// Mitsubishi GX Works2 project: Group12_PLC s (3)   PLC: FX3G

// global labels: Global1
VAR_GLOBAL
  startSwitch AT X007 : BOOL;
  initBisuit AT D1100 : REAL;
END_VAR
VAR_GLOBAL CONSTANT
  sixBis : REAL := 6.0;
END_VAR
VAR_GLOBAL
  enoughBuscuits AT M0 : BOOL;
  initCream AT D1102 : REAL;
END_VAR
VAR_GLOBAL CONSTANT
  threeHunCream : REAL := 300.0;
END_VAR
VAR_GLOBAL
  enoughCream AT M1 : BOOL;
  initChoclate AT D1104 : REAL;
END_VAR
VAR_GLOBAL CONSTANT
  twofourtyCho : REAL := 240.0;
END_VAR
VAR_GLOBAL
  enoughCoclate AT M2 : BOOL;
  startWday AT Y007 : BOOL;
  storeBuscuit AT D1106 : REAL;
  storeCream AT D1108 : REAL;
  storeChoclate AT D1110 : REAL;
  WD_started AT M40 : BOOL;
  FP_QA AT Y003 : BOOL;
  closeDay_HL AT M3 : BOOL;
  check AT M4 : BOOL;
  blink AT M4 : BOOL;
  activeDay AT Y007 : BOOL;
  stop3sec AT M5 : BOOL;
  activeDay_LI AT Y007 : BOOL;
  endBlink AT M6 : BOOL;
  finishing AT M60 : BOOL;
END_VAR
VAR_GLOBAL CONSTANT
  zeroCon : REAL;
END_VAR
VAR_GLOBAL
  stCounter AT CC1 : BOOL;
  scndCounter AT CC2 : BOOL;
  perfusion AT D1111 : REAL;
  Cream_perfusion AT D1112 : REAL;
  surfaceA AT D1114 : REAL;
  surfaceb AT D1116 : REAL;
  readyKrimbo AT D1118 : REAL;
  enoughBuscuitsTo_GoOn AT M10 : BOOL;
  enoughCreamTo_GoOn AT M11 : BOOL;
  enoughCoclateTo_GoOn AT M12 : BOOL;
  enoughStore AT M80 : BOOL;
  Ziluf_switch AT X011 : BOOL;
  ZilufContiner AT D1112 : REAL;
  moveToZiluf AT M90 : BOOL;
  moveTo_Ziluf AT M90 : BOOL;
  Machinestart_switchA AT X010 : BOOL;
  Carambosurface AT X001 : BOOL;
  Sprinkling_performed AT X003 : BOOL;
  TempAbove30 AT X030 : BOOL;
  TempLower15 AT X015 : BOOL;
  Sprinkling_isOn AT Y010 : BOOL;
  Machine_lampA AT Y004 : BOOL;
  faultIs_detected AT X002 : BOOL;
  stopMachine AT X005 : BOOL;
  ziluf_isOn AT Y010 : BOOL;
  krimboSurface AT X001 : BOOL;
END_VAR
VAR_GLOBAL CONSTANT
  subCream300 : REAL := 300.0;
  subBisctuit : REAL := 6.0;
END_VAR
VAR_GLOBAL
  Machine_lampAOn AT Y004 : BOOL;
  perfusion_performed AT X003 : BOOL;
  MachineA AT Y004 : BOOL;
  MachineA_off AT Y004 : BOOL;
  Machine_lampAoff AT X005 : BOOL;
  imageProcessing AT X003 : BOOL;
  perfusion_lampA AT Y004 : BOOL;
  perfusion_lampAOn AT Y004 : BOOL;
  perfusion_lampAoff AT X005 : BOOL;
  perfusion_switchA AT X010 : BOOL;
  Transportation AT M13 : BOOL;
  Timer4 AT TC4 : BOOL;
END_VAR
VAR_GLOBAL CONSTANT
  four_seconds : INT := 40;
END_VAR
VAR_GLOBAL
  output_Timer4 AT TS4 : BOOL;
  output_Timer3 AT TS4 : BOOL;
  output_Timer1 AT TS1 : BOOL;
  blinking_Input AT M14 : BOOL;
END_VAR
VAR_GLOBAL CONSTANT
  half_Second : INT := 5;
END_VAR
VAR_GLOBAL
  Timer2 AT TC0 : BOOL;
  Timer0 AT TC0 : BOOL;
  output_Timer0 AT TS0 : BOOL;
  Trans_Lamp0 AT Y000 : BOOL;
  Timer1 AT TC1 : BOOL;
  Trans_Lamp1 AT Y001 : BOOL;
  end_Tranportation AT M15 : BOOL;
  endTranportation AT M15 : BOOL;
  startFroasting AT X006 : BOOL;
  start_Froasting AT X006 : BOOL;
  AnalogInput1 AT D8280 : INT;
  save_Analog_Value AT D1114 : INT;
END_VAR
VAR_GLOBAL CONSTANT
  realUnit : INT := 400;
  ConstFive : INT := 5;
END_VAR
VAR_GLOBAL
  normalFroasting AT M16 : BOOL;
END_VAR
VAR_GLOBAL CONSTANT
  ConstTen : INT := 10;
END_VAR
VAR_GLOBAL
  less_thanTen : BOOL;
END_VAR
VAR_GLOBAL CONSTANT
  ConstSex : INT := 6;
  ConstSix : INT := 6;
END_VAR
VAR_GLOBAL
  doubleFroasting AT M17 : BOOL;
END_VAR
VAR_GLOBAL CONSTANT
  Chocolate_normalAmount : REAL := 120.0;
  Chocolate_normalAmount120 : REAL := 120.0;
END_VAR
VAR_GLOBAL
  Chocolate_in_process AT D1116 : REAL;
END_VAR
VAR_GLOBAL CONSTANT
  Chocolate_normalAmount240 : REAL := 240.0;
  Chocolate_doubleAmount240 : REAL := 240.0;
END_VAR
VAR_GLOBAL
  Finished_normalChocolateProcess AT M18 : BOOL;
  Finished_doubleChocolateProcess AT M19 : BOOL;
  Timer5 AT TC5 : BOOL;
END_VAR
VAR_GLOBAL CONSTANT
  five_seconds : INT := 50;
END_VAR
VAR_GLOBAL
  Froasting_Timer AT TS5 : BOOL;
  Froasting_Lamp AT Y003 : BOOL;
  startPackaging_krimbo AT X000 : BOOL;
  startCounter5_krimpo AT CC5 : BOOL;
END_VAR
VAR_GLOBAL CONSTANT
  Five_units : INT := 5;
END_VAR
VAR_GLOBAL
  finish_counter AT CS1 : BOOL;
END_VAR
VAR_GLOBAL CONSTANT
  six_units : INT := 6;
END_VAR
VAR_GLOBAL
  end_counting AT CC22 : BOOL;
  finish_packaging AT M20 : BOOL;
  end_countingPackaged AT CC6 : BOOL;
  end_packaging AT CS2 : BOOL;
  packagingLamp AT Y002 : BOOL;
  Add_6Krimbo AT D8280 : INT;
  krimbos_quantity AT D1118 : INT;
  start_WorkDay AT X007 : BOOL;
  end_DayBlink AT M66 : BOOL;
  blink_Seconds AT TC3 : BOOL;
END_VAR
VAR_GLOBAL CONSTANT
  threeSeconds : INT := 30;
END_VAR
VAR_GLOBAL
  blink_Timer AT TS3 : BOOL;
  blink_timeH AT M90 : BOOL;
  blink_stCounter AT TC7 : BOOL;
END_VAR
VAR_GLOBAL CONSTANT
  halfConst : INT := 5;
END_VAR
VAR_GLOBAL
  stBlink AT M61 : BOOL;
  stBlinkingTime AT TS7 : BOOL;
  st_blink AT M62 : BOOL;
  blink_scndCounter AT TC8 : BOOL;
  scnd_blink AT M63 : BOOL;
  scndBlinkingTime AT TS8 : BOOL;
  WD_ended AT M67 : BOOL;
  help1 AT M77 : BOOL;
END_VAR

// task Task_01 (event TRUE, interval 0, priority 31): POU_01

PROGRAM POU_01
(* structured ladder/FBD written out as ST: instructions are called as NAME(EN, inputs, outputs); _pN, _eN, _tN stand for wires *)
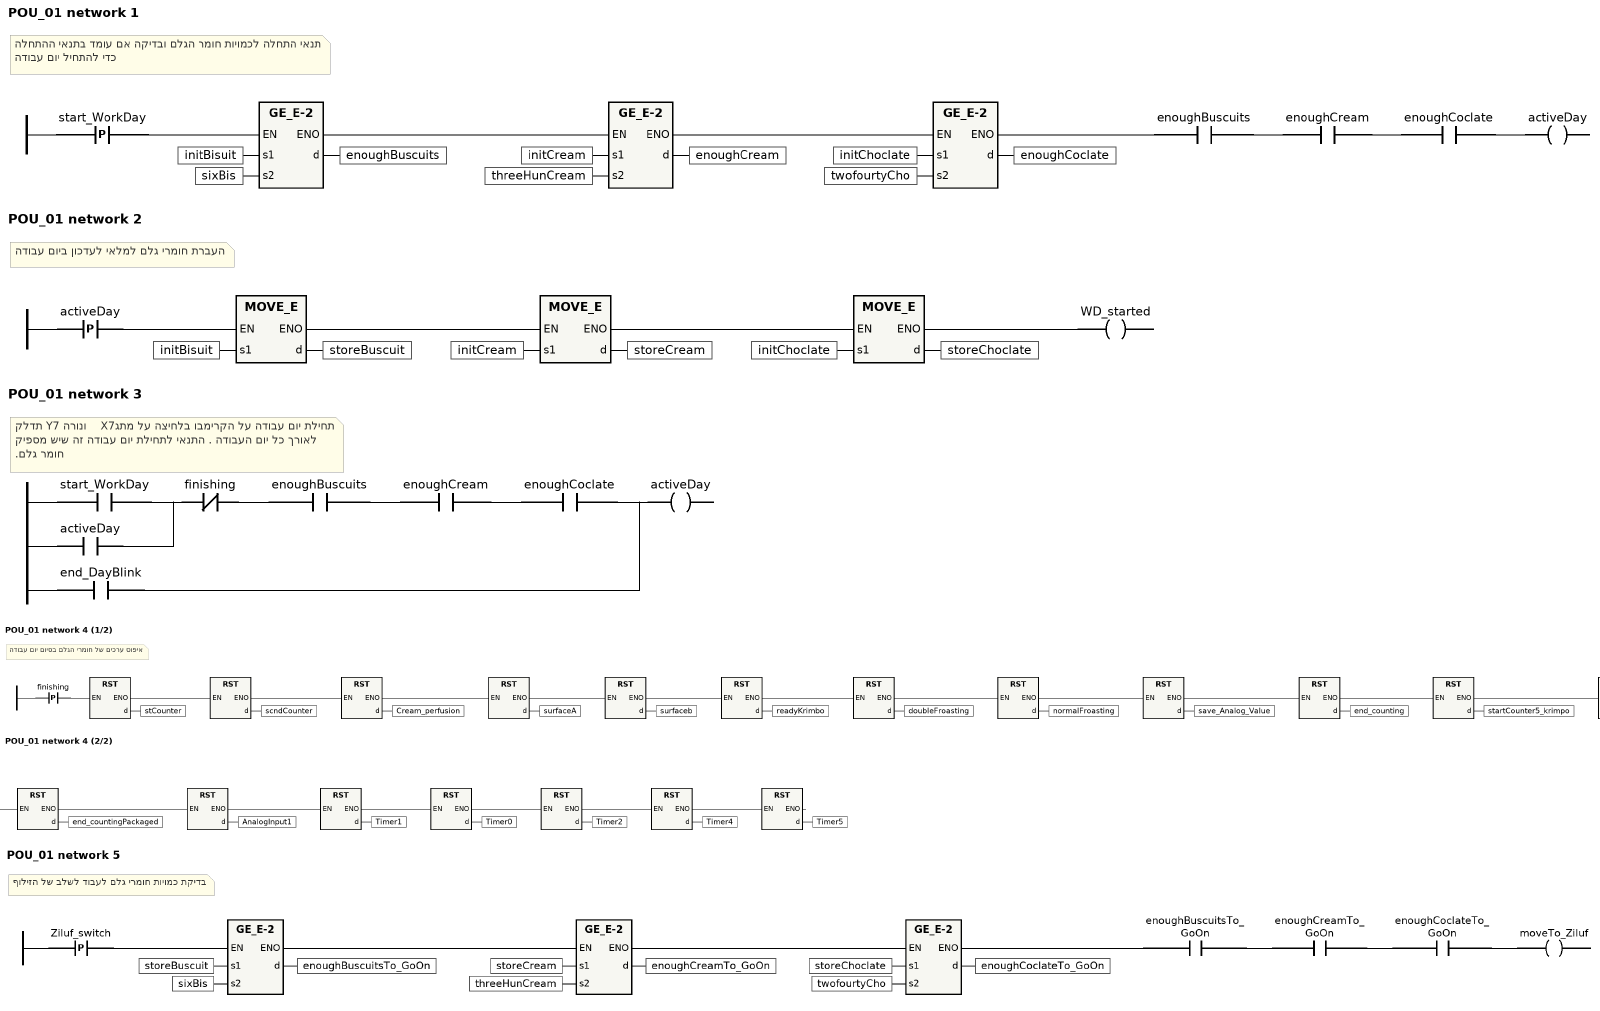
(* network 1 *)
(* תנאי התחלה לכמויות חומר הגלם ובדיקה אם עומד בתנאי ההתחלה כדי להתחיל יום עבודה *)
_e1 := GE_E(LDP(TRUE, start_WorkDay), initBisuit, sixBis, enoughBuscuits);
_e2 := GE_E(_e1, initCream, threeHunCream, enoughCream);
_e3 := GE_E(_e2, initChoclate, twofourtyCho, enoughCoclate);
activeDay := _e3 AND enoughBuscuits AND enoughCream AND enoughCoclate;
(* network 2 *)
(* העברת חומרי גלם למלאי לעדכון ביום עבודה *)
_e1 := MOVE_E(LDP(TRUE, activeDay), initBisuit, storeBuscuit);
_e2 := MOVE_E(_e1, initCream, storeCream);
_e3 := MOVE_E(_e2, initChoclate, storeChoclate);
WD_started := _e3;
(* network 3 *)
(* תחילת יום עבודה על הקרימבו בלחיצה על מתגX7    ונורה Y7 תדלק לאורך כל יום העבודה . התנאי לתחילת יום עבודה זה שיש מספיק חומר גלם. *)
activeDay := (((((start_WorkDay OR activeDay) AND NOT finishing) AND enoughBuscuits) AND enoughCream) AND enoughCoclate) OR end_DayBlink;
(* network 4 *)
(* איפוס ערכים של חומרי הגלם בסיום יום עבודה *)
_e1 := RST(LDP(TRUE, finishing), stCounter);
_e2 := RST(_e1, scndCounter);
_e3 := RST(_e2, Cream_perfusion);
_e4 := RST(_e3, surfaceA);
_e5 := RST(_e4, surfaceb);
_e6 := RST(_e5, readyKrimbo);
_e7 := RST(_e6, doubleFroasting);
_e8 := RST(_e7, normalFroasting);
_e9 := RST(_e8, save_Analog_Value);
_e10 := RST(_e9, end_counting);
_e11 := RST(_e10, startCounter5_krimpo);
_e12 := RST(_e11, end_countingPackaged);
_e13 := RST(_e12, AnalogInput1);
_e14 := RST(_e13, Timer1);
_e15 := RST(_e14, Timer0);
_e16 := RST(_e15, Timer2);
_e17 := RST(_e16, Timer4);
RST(_e17, Timer5);
(* network 5 *)
(* בדיקת כמויות חומרי גלם לעבוד לשלב של הזילוף *)
_e1 := GE_E(LDP(TRUE, Ziluf_switch), storeBuscuit, sixBis, enoughBuscuitsTo_GoOn);
_e2 := GE_E(_e1, storeCream, threeHunCream, enoughCreamTo_GoOn);
_e3 := GE_E(_e2, storeChoclate, twofourtyCho, enoughCoclateTo_GoOn);
moveTo_Ziluf := _e3 AND enoughBuscuitsTo_GoOn AND enoughCreamTo_GoOn AND enoughCoclateTo_GoOn;
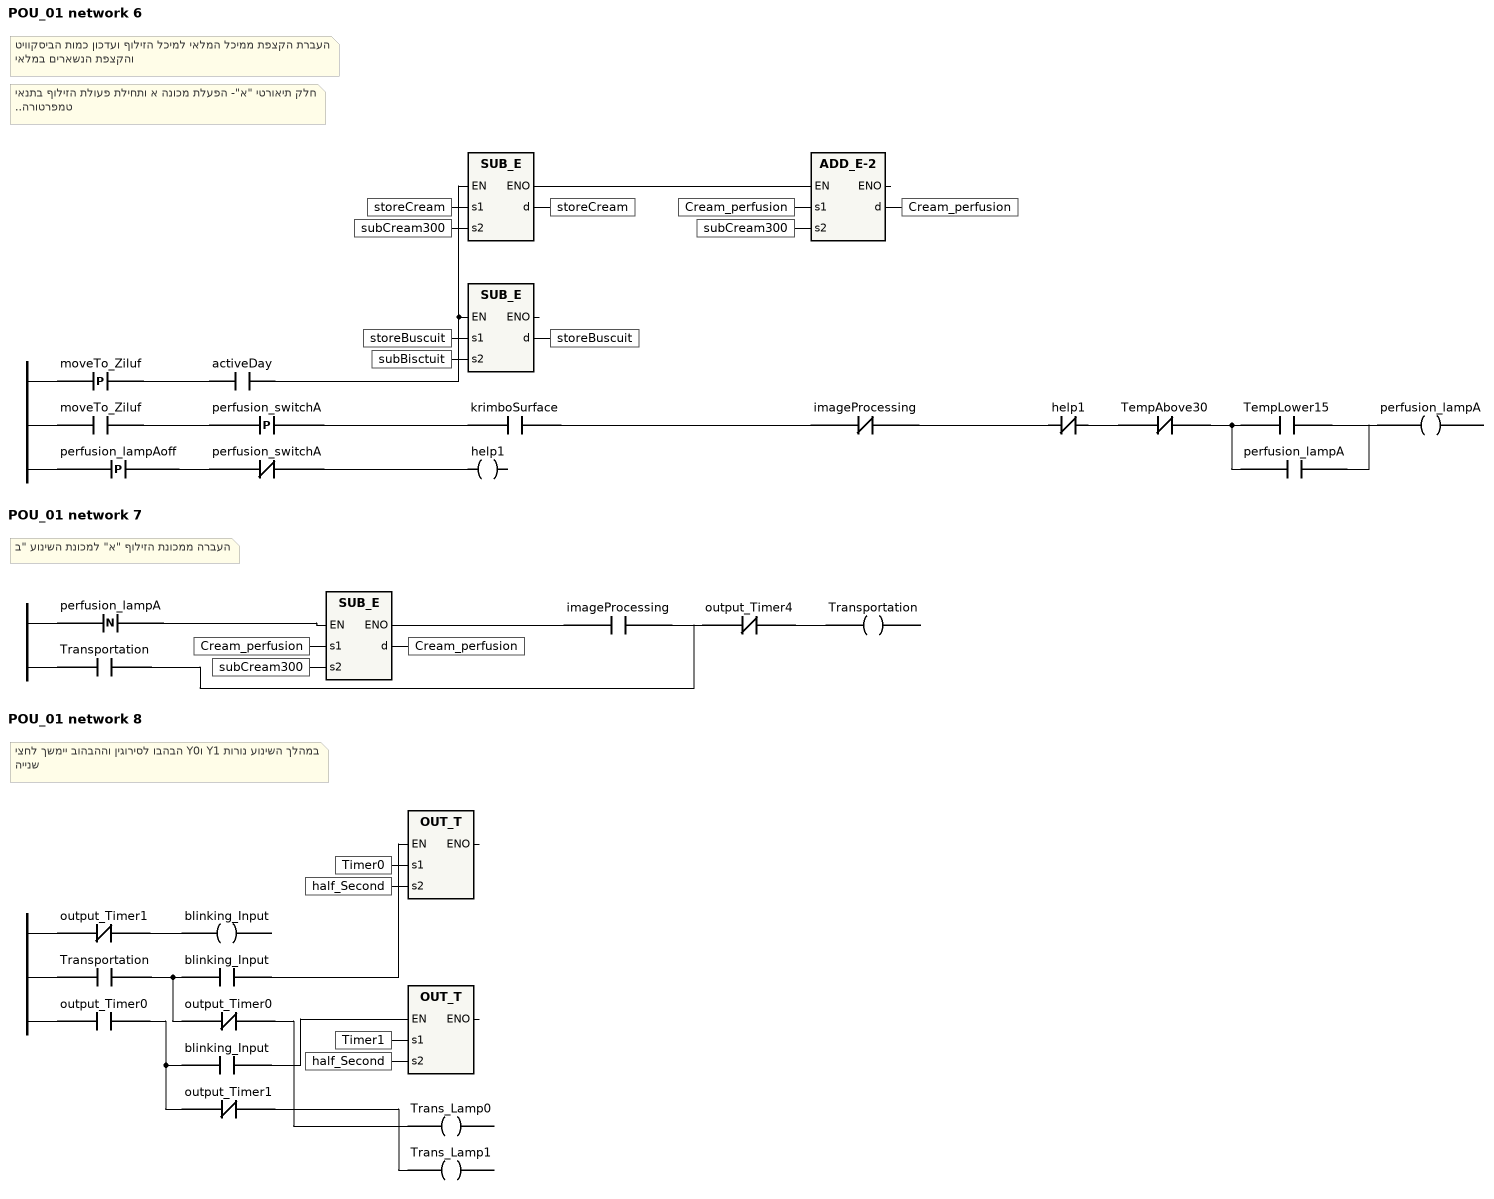
(* network 6 *)
(* העברת הקצפת ממיכל המלאי למיכל הזילוף ועדכון כמות הביסקוויט והקצפת הנשארים במלאי *)
(* חלק תיאורטי "א"- הפעלת מכונה א ותחילת פעולת הזילוף בתנאי טמפרטורה.. *)
_p1 := LDP(TRUE, moveTo_Ziluf) AND activeDay;
_e2 := SUB_E(_p1, storeCream, subCream300, storeCream);
ADD_E(_e2, Cream_perfusion, subCream300, Cream_perfusion);
SUB_E(_p1, storeBuscuit, subBisctuit, storeBuscuit);
_p3 := moveTo_Ziluf AND LDP(TRUE, perfusion_switchA) AND krimboSurface AND NOT imageProcessing AND NOT help1 AND NOT TempAbove30;
perfusion_lampA := (_p3 AND TempLower15) OR (_p3 AND perfusion_lampA);
help1 := LDP(TRUE, perfusion_lampAoff) AND NOT perfusion_switchA;
(* network 7 *)
(* העברה ממכונת הזילוף "א" למכונת השינוע "ב *)
_e1 := SUB_E(LDF(TRUE, perfusion_lampA), Cream_perfusion, subCream300, Cream_perfusion);
Transportation := ((_e1 AND imageProcessing) OR Transportation) AND NOT output_Timer4;
(* network 8 *)
(* במהלך השינוע נורות Y1 וY0 הבהבו לסירוגין וההבהוב יימשך לחצי שנייה *)
blinking_Input := NOT output_Timer1;
OUT_T(Transportation AND blinking_Input, Timer0, half_Second);
Trans_Lamp0 := Transportation AND NOT output_Timer0;
OUT_T(output_Timer0 AND blinking_Input, Timer1, half_Second);
Trans_Lamp1 := output_Timer0 AND NOT output_Timer1;
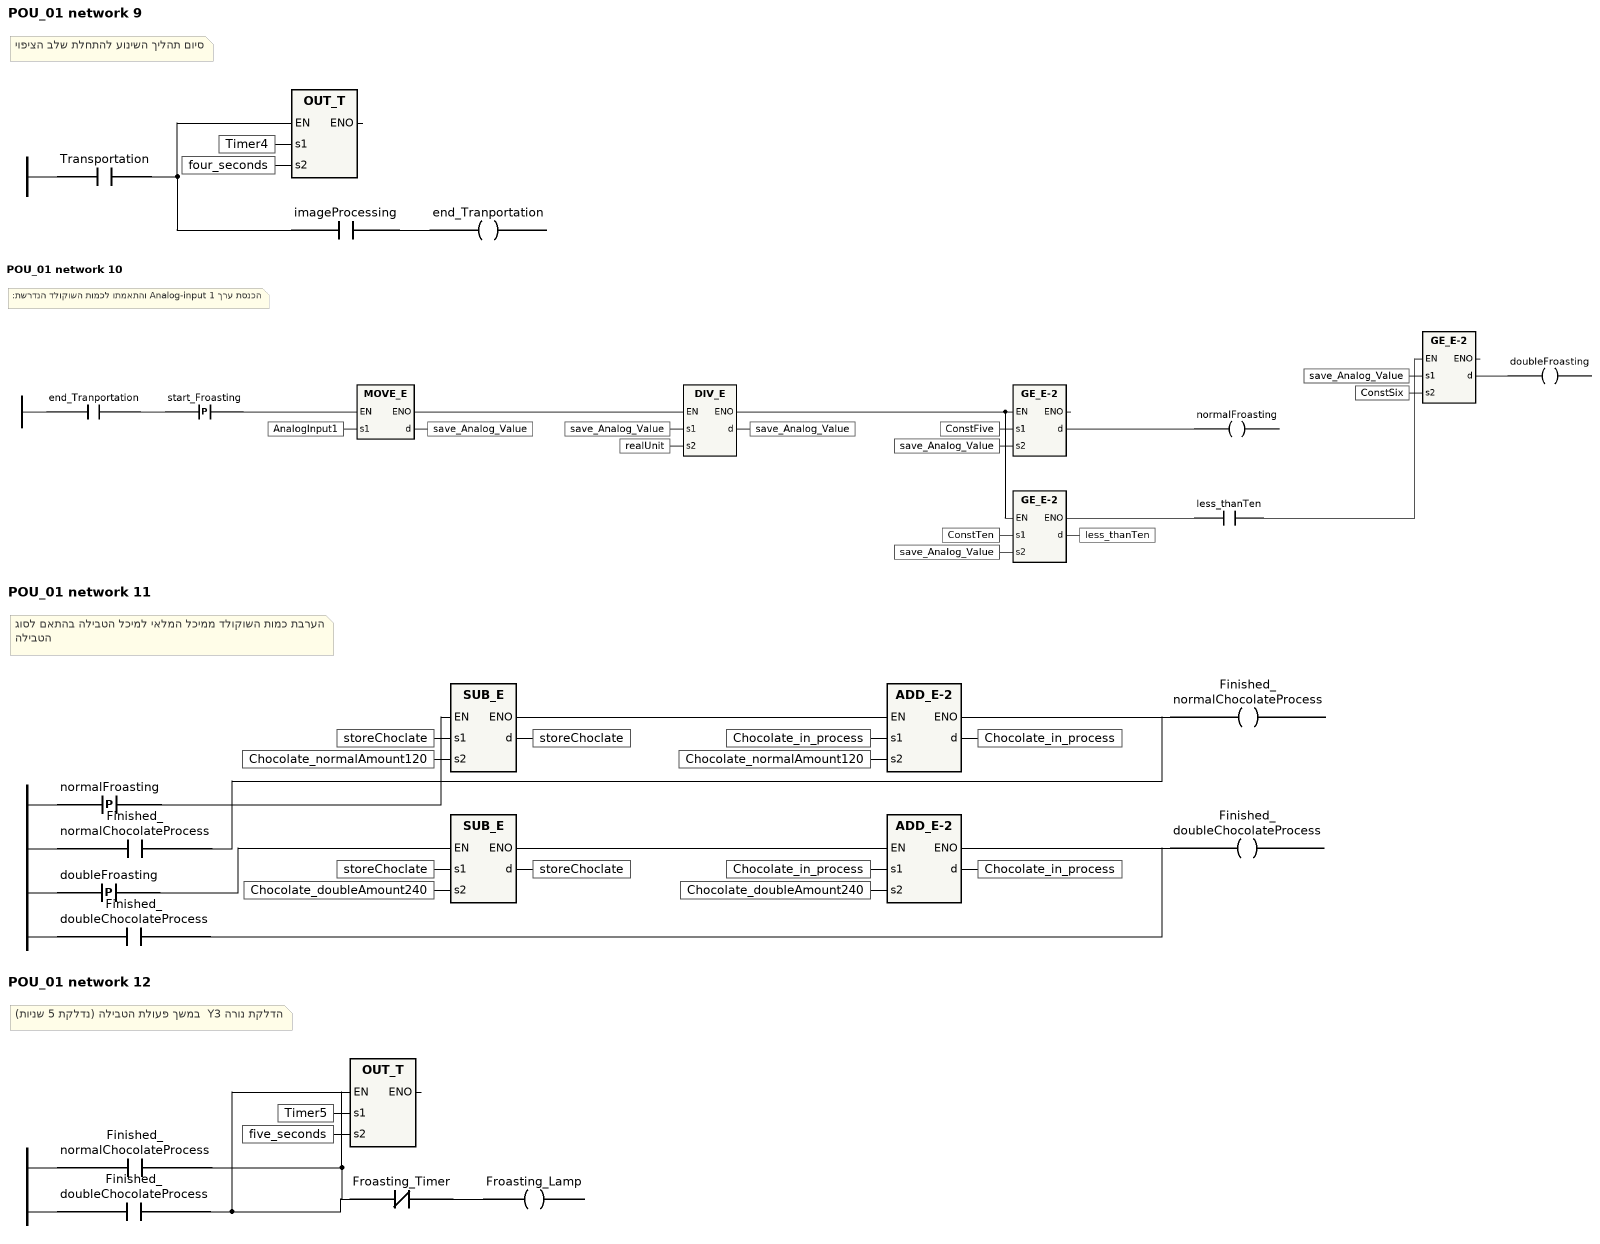
(* network 9 *)
(* סיום תהליך השינוע להתחלת שלב הציפוי *)
OUT_T(Transportation, Timer4, four_seconds);
end_Tranportation := Transportation AND imageProcessing;
(* network 10 *)
(* הכנסת ערך Analog-input 1 והתאמתו לכמות השוקולד הנדרשת: *)
_e1 := MOVE_E(end_Tranportation AND LDP(TRUE, start_Froasting), AnalogInput1, save_Analog_Value);
_e2 := DIV_E(_e1, save_Analog_Value, realUnit, save_Analog_Value);
GE_E(_e2, ConstFive, save_Analog_Value, _t3);
normalFroasting := _t3;
_e4 := GE_E(_e2, ConstTen, save_Analog_Value, less_thanTen);
GE_E(_e4 AND less_thanTen, save_Analog_Value, ConstSix, _t5);
doubleFroasting := _t5;
(* network 11 *)
(* הערבת כמות השוקולד ממיכל המלאי למיכל הטבילה בהתאם לסוג הטבילה *)
_e1 := SUB_E(LDP(TRUE, normalFroasting), storeChoclate, Chocolate_normalAmount120, storeChoclate);
_e2 := ADD_E(_e1, Chocolate_in_process, Chocolate_normalAmount120, Chocolate_in_process);
Finished_normalChocolateProcess := _e2 OR Finished_normalChocolateProcess;
_e3 := SUB_E(LDP(TRUE, doubleFroasting), storeChoclate, Chocolate_doubleAmount240, storeChoclate);
_e4 := ADD_E(_e3, Chocolate_in_process, Chocolate_doubleAmount240, Chocolate_in_process);
Finished_doubleChocolateProcess := _e4 OR Finished_doubleChocolateProcess;
(* network 12 *)
(* הדלקת נורה Y3  במשך פעולת הטבילה (נדלקת 5 שניות) *)
_p1 := Finished_normalChocolateProcess OR Finished_doubleChocolateProcess;
OUT_T(_p1, Timer5, five_seconds);
Froasting_Lamp := _p1 AND NOT Froasting_Timer;
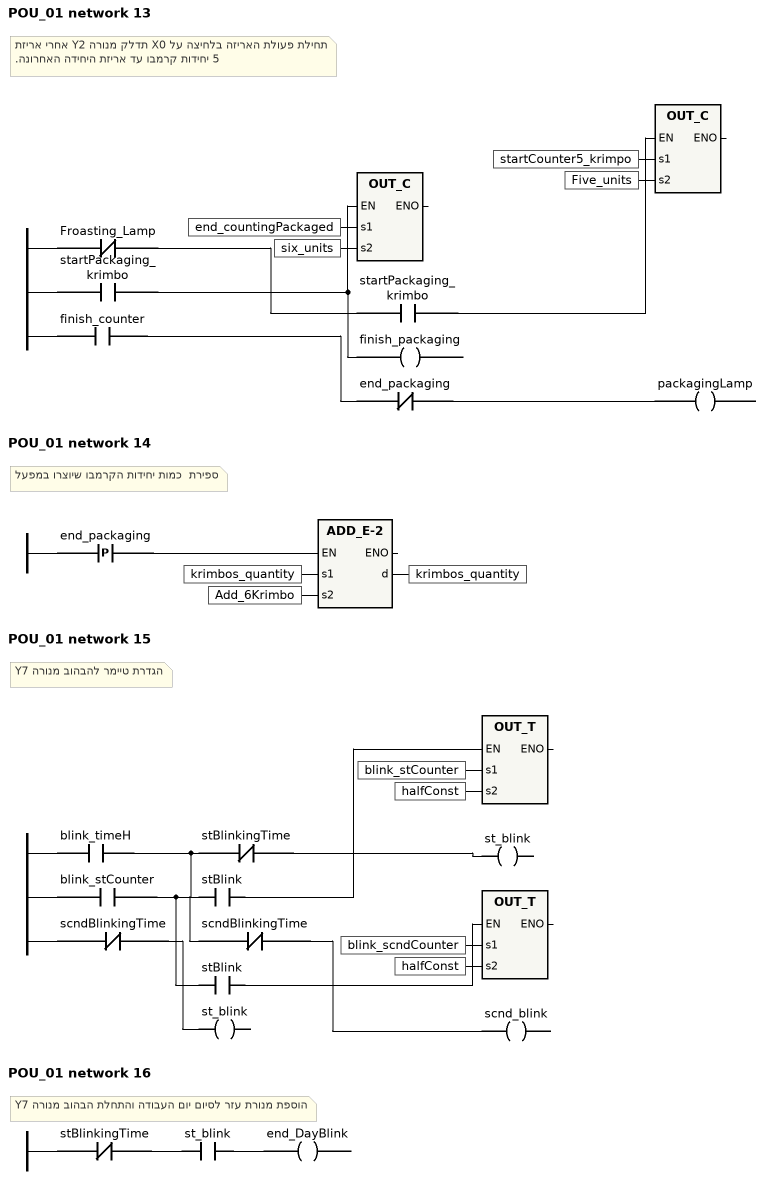
(* network 13 *)
(* תחילת פעולת האריזה בלחיצה על X0 תדלק מנורה Y2 אחרי אריזת 5 יחידות קרמבו עד אריזת היחידה האחרונה. *)
OUT_C(NOT Froasting_Lamp AND startPackaging_krimbo, startCounter5_krimpo, Five_units);
OUT_C(startPackaging_krimbo, end_countingPackaged, six_units);
finish_packaging := startPackaging_krimbo;
packagingLamp := finish_counter AND NOT end_packaging;
(* network 14 *)
(* ספירת  כמות יחידות הקרמבו שיוצרו במפעל *)
ADD_E(LDP(TRUE, end_packaging), krimbos_quantity, Add_6Krimbo, krimbos_quantity);
(* network 15 *)
(* הגדרת טיימר להבהוב מנורה Y7 *)
st_blink := blink_timeH AND NOT stBlinkingTime;
OUT_T(blink_timeH AND stBlink, blink_stCounter, halfConst);
scnd_blink := blink_stCounter AND NOT scndBlinkingTime;
OUT_T(blink_stCounter AND stBlink, blink_scndCounter, halfConst);
st_blink := NOT scndBlinkingTime;
(* network 16 *)
(* הוספת מנורת עזר לסיום יום העבודה והתחלת הבהוב מנורה Y7 *)
end_DayBlink := NOT stBlinkingTime AND st_blink;
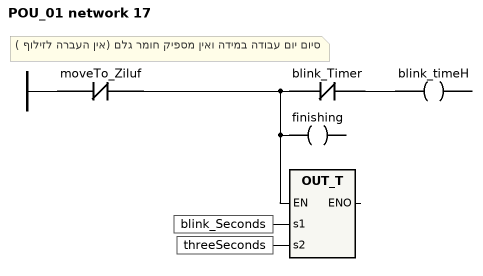
(* network 17 *)
(* סיום יום עבודה במידה ואין מספיק חומר גלם (אין העברה לזילוף ) *)
_p1 := NOT moveTo_Ziluf;
blink_timeH := _p1 AND NOT blink_Timer;
finishing := _p1;
OUT_T(_p1, blink_Seconds, threeSeconds);
END_PROGRAM
